LIN {X 0,Y 106.006,Z 264.737,A -85,B 0,C 180,E1 -28471.398,E2 -28471.398} C_VEL
LIN {X 0,Y 102.462,Z 273.009,A -85,B 0,C 180,E1 -28472.836,E2 -28472.836} C_VEL
LIN {X 0,Y 98.379,Z 281.013,A -85,B 0,C 180,E1 -28474.767,E2 -28474.767} C_VEL
LIN {X 0,Y 93.024,Z 289.74,A -85,B 0,C 180,E1 -28477.584,E2 -28477.584} C_VEL
LIN {X 0,Y 86.706,Z 298.118,A -85,B 0,C 180,E1 -28481.432,E2 -28481.432} C_VEL
LIN {X 0,Y 82.048,Z 303.608,A -85,B 0,C 180,E1 -28485.037,E2 -28485.037} C_VEL
LIN {X 0,Y 76.639,Z 309.153,A -85,B 0,C 180,E1 -28490.067,E2 -28490.067} C_VEL
LIN {X 0,Y 71.093,Z 314.313,A -85,B 0,C 180,E1 -28497.065,E2 -28497.065} C_VEL
LIN {X 0,Y 66.84,Z 318.102,A -85,B 0,C 180,E1 -28505.13,E2 -28505.13} C_VEL
LIN {X 0,Y 64.768,Z 319.84,A -85,B 0,C 180,E1 -28511.004,E2 -28511.004} C_VEL
LIN {X 0,Y 63.342,Z 321.084,A -85,B 0,C 180,E1 -28517.181,E2 -28517.181} C_VEL
LIN {X 0,Y 62.596,Z 321.855,A -85,B 0,C 180,E1 -28523.555,E2 -28523.555} C_VEL
LIN {X 0,Y 62.546,Z 322.148,A -85,B 0,C 180,E1 -28530.002,E2 -28530.002} C_VEL
LIN {X 0,Y 62.595,Z 321.84,A -85,B 0,C 180,E1 -28536.448,E2 -28536.448} C_VEL
LIN {X 0,Y 63.338,Z 321.04,A -85,B 0,C 180,E1 -28542.823,E2 -28542.823} C_VEL
LIN {X 0,Y 64.752,Z 319.768,A -85,B 0,C 180,E1 -28549.004,E2 -28549.004} C_VEL
LIN {X 0,Y 68.103,Z 316.843,A -85,B 0,C 180,E1 -28557.672,E2 -28557.672} C_VEL
LIN {X 0,Y 71.086,Z 314.178,A -85,B 0,C 180,E1 -28562.942,E2 -28562.942} C_VEL
LIN {X 0,Y 76.621,Z 308.98,A -85,B 0,C 180,E1 -28569.948,E2 -28569.948} C_VEL
LIN {X 0,Y 83.174,Z 302.123,A -85,B 0,C 180,E1 -28575.91,E2 -28575.91} C_VEL
LIN {X 0,Y 89.214,Z 294.637,A -85,B 0,C 180,E1 -28580.183,E2 -28580.183} C_VEL
LIN {X 0,Y 94.643,Z 286.803,A -85,B 0,C 180,E1 -28583.357,E2 -28583.357} C_VEL
LIN {X 0,Y 98.847,Z 279.71,A -85,B 0,C 180,E1 -28585.475,E2 -28585.475} C_VEL
LIN {X 0,Y 103.176,Z 270.972,A -85,B 0,C 180,E1 -28587.454,E2 -28587.454} C_VEL
LIN {X 0,Y 107.193,Z 260.903,A -85,B 0,C 180,E1 -28589.085,E2 -28589.085} C_VEL
LIN {X 0,Y 110.412,Z 249.756,A -85,B 0,C 180,E1 -28590.251,E2 -28590.251} C_VEL
LIN {X 0,Y 112.274,Z 240.076,A -85,B 0,C 180,E1 -28590.927,E2 -28590.927} C_VEL
LIN {X 0,Y 112.893,Z 234.742,A -85,B 0,C 180,E1 -28591.299,E2 -28591.299} C_VEL
LIN {X 0,Y 110.571,Z 229.113,A -85,B 0,C 180,E1 -28594.385,E2 -28594.385} C_VEL
LIN {X 0,Y 107.513,Z 222.914,A -85,B 0,C 180,E1 -28599.102,E2 -28599.102} C_VEL
LIN {X 0,Y 105.679,Z 219.605,A -85,B 0,C 180,E1 -28602.574,E2 -28602.574} C_VEL
LIN {X 0,Y 103.849,Z 216.166,A -85,B 0,C 180,E1 -28607.104,E2 -28607.104} C_VEL
LIN {X 0,Y 102.285,Z 213.382,A -85,B 0,C 180,E1 -28613.094,E2 -28613.094} C_VEL
LIN {X 0,Y 101.962,Z 211.83,A -85,B 0,C 180,E1 -28616.048,E2 -28616.048} C_VEL
LIN {X 0,Y 101.746,Z 211.461,A -85,B 0,C 180,E1 -28620,E2 -28620} C_VEL
LIN {X 0,Y 102.06,Z 212.11,A -85,B 0,C 180,E1 -28625.186,E2 -28625.186} C_VEL
LIN {X 0,Y 103.108,Z 215.279,A -85,B 0,C 180,E1 -28630.962,E2 -28630.962} C_VEL
LIN {X 0,Y 104.122,Z 216.678,A -85,B 0,C 180,E1 -28633.975,E2 -28633.975} C_VEL
LIN {X 0,Y 106.566,Z 221.249,A -85,B 0,C 180,E1 -28639.504,E2 -28639.504} C_VEL
LIN {X 0,Y 109.022,Z 225.911,A -85,B 0,C 180,E1 -28643.66,E2 -28643.66} C_VEL
LIN {X 0,Y 111.679,Z 231.652,A -85,B 0,C 180,E1 -28647.42,E2 -28647.42} C_VEL
LIN {X 0,Y 111.991,Z 233.692,A -85,B 0,C 180,E1 -28648.036,E2 -28648.036} C_VEL
LIN {X 0,Y 111.67,Z 236.769,A -85,B 0,C 180,E1 -28648.253,E2 -28648.253} C_VEL
LIN {X 0,Y 110.414,Z 241.191,A -85,B 0,C 180,E1 -28647.938,E2 -28647.938} C_VEL
LIN {X 0,Y 107.648,Z 248.027,A -85,B 0,C 180,E1 -28647.095,E2 -28647.095} C_VEL
LIN {X 0,Y 106.129,Z 252.208,A -85,B 0,C 180,E1 -28647.118,E2 -28647.118} C_VEL
LIN {X 0,Y 102.863,Z 261.996,A -85,B 0,C 180,E1 -28648.34,E2 -28648.34} C_VEL
LIN {X 0,Y 99.46,Z 270.01,A -85,B 0,C 180,E1 -28649.711,E2 -28649.711} C_VEL
LIN {X 0,Y 95.68,Z 277.368,A -85,B 0,C 180,E1 -28651.361,E2 -28651.361} C_VEL
LIN {X 0,Y 90.795,Z 285.27,A -85,B 0,C 180,E1 -28653.682,E2 -28653.682} C_VEL
LIN {X 0,Y 86.772,Z 290.94,A -85,B 0,C 180,E1 -28655.908,E2 -28655.908} C_VEL
LIN {X 0,Y 81.521,Z 297.279,A -85,B 0,C 180,E1 -28659.112,E2 -28659.112} C_VEL
LIN {X 0,Y 76.576,Z 302.546,A -85,B 0,C 180,E1 -28662.757,E2 -28662.757} C_VEL
LIN {X 0,Y 71.98,Z 306.943,A -85,B 0,C 180,E1 -28666.883,E2 -28666.883} C_VEL
LIN {X 0,Y 65.955,Z 312.112,A -85,B 0,C 180,E1 -28674.12,E2 -28674.12} C_VEL
LIN {X 0,Y 62.546,Z 314.761,A -85,B 0,C 180,E1 -28679.624,E2 -28679.624} C_VEL
LIN {X 0,Y 58.603,Z 317.66,A -85,B 0,C 180,E1 -28688.912,E2 -28688.912} C_VEL
LIN {X 0,Y 56.87,Z 318.92,A -85,B 0,C 180,E1 -28695.689,E2 -28695.689} C_VEL
LIN {X 0,Y 55.802,Z 319.711,A -85,B 0,C 180,E1 -28702.763,E2 -28702.763} C_VEL
LIN {X 0,Y 55.488,Z 320.012,A -85,B 0,C 180,E1 -28709.998,E2 -28709.998} C_VEL
LIN {X 0,Y 55.796,Z 319.73,A -85,B 0,C 180,E1 -28717.234,E2 -28717.234} C_VEL
LIN {X 0,Y 56.831,Z 318.976,A -85,B 0,C 180,E1 -28724.318,E2 -28724.318} C_VEL
LIN {X 0,Y 58.588,Z 317.754,A -85,B 0,C 180,E1 -28731.09,E2 -28731.09} C_VEL
LIN {X 0,Y 62.5,Z 314.894,A -85,B 0,C 180,E1 -28740.397,E2 -28740.397} C_VEL
LIN {X 0,Y 65.894,Z 312.287,A -85,B 0,C 180,E1 -28745.915,E2 -28745.915} C_VEL
LIN {X 0,Y 71.932,Z 307.164,A -85,B 0,C 180,E1 -28753.149,E2 -28753.149} C_VEL
LIN {X 0,Y 77.728,Z 301.649,A -85,B 0,C 180,E1 -28758.238,E2 -28758.238} C_VEL
LIN {X 0,Y 84.044,Z 294.711,A -85,B 0,C 180,E1 -28762.598,E2 -28762.598} C_VEL
LIN {X 0,Y 90.063,Z 286.746,A -85,B 0,C 180,E1 -28766.006,E2 -28766.006} C_VEL
LIN {X 0,Y 94.945,Z 279.15,A -85,B 0,C 180,E1 -28768.346,E2 -28768.346} C_VEL
LIN {X 0,Y 99.362,Z 270.874,A -85,B 0,C 180,E1 -28770.257,E2 -28770.257} C_VEL
LIN {X 0,Y 102.782,Z 263.051,A -85,B 0,C 180,E1 -28771.623,E2 -28771.623} C_VEL
LIN {X 0,Y 105.714,Z 254.557,A -85,B 0,C 180,E1 -28772.773,E2 -28772.773} C_VEL
LIN {X 0,Y 108.126,Z 245.305,A -85,B 0,C 180,E1 -28773.657,E2 -28773.657} C_VEL
LIN {X 0,Y 109.418,Z 238.026,A -85,B 0,C 180,E1 -28774.203,E2 -28774.203} C_VEL
LIN {X 0,Y 107.073,Z 231.956,A -85,B 0,C 180,E1 -28778.341,E2 -28778.341} C_VEL
LIN {X 0,Y 104.905,Z 227.419,A -85,B 0,C 180,E1 -28782.564,E2 -28782.564} C_VEL
LIN {X 0,Y 102.825,Z 223.047,A -85,B 0,C 180,E1 -28788.167,E2 -28788.167} C_VEL
LIN {X 0,Y 101.53,Z 220.472,A -85,B 0,C 180,E1 -28794.009,E2 -28794.009} C_VEL
LIN {X 0,Y 101.307,Z 218.967,A -85,B 0,C 180,E1 -28797.017,E2 -28797.017} C_VEL
LIN {X 0,Y 101.224,Z 218.755,A -85,B 0,C 180,E1 -28800.994,E2 -28800.994} C_VEL
LIN {X 0,Y 101.361,Z 219.335,A -85,B 0,C 180,E1 -28803.727,E2 -28803.727} C_VEL
LIN {X 0,Y 102.513,Z 222.681,A -85,B 0,C 180,E1 -28810.617,E2 -28810.617} C_VEL
LIN {X 0,Y 103.083,Z 223.715,A -85,B 0,C 180,E1 -28812.504,E2 -28812.504} C_VEL
LIN {X 0,Y 105.017,Z 227.64,A -85,B 0,C 180,E1 -28817.471,E2 -28817.471} C_VEL
LIN {X 0,Y 107.183,Z 232.16,A -85,B 0,C 180,E1 -28821.634,E2 -28821.634} C_VEL
LIN {X 0,Y 109.493,Z 238.014,A -85,B 0,C 180,E1 -28825.569,E2 -28825.569} C_VEL
LIN {X 0,Y 108.088,Z 246.375,A -85,B 0,C 180,E1 -28826.138,E2 -28826.138} C_VEL
LIN {X 0,Y 105.582,Z 255.84,A -85,B 0,C 180,E1 -28826.934,E2 -28826.934} C_VEL
LIN {X 0,Y 102.486,Z 264.614,A -85,B 0,C 180,E1 -28828.007,E2 -28828.007} C_VEL
LIN {X 0,Y 98.787,Z 272.886,A -85,B 0,C 180,E1 -28829.369,E2 -28829.369} C_VEL
LIN {X 0,Y 94.502,Z 280.888,A -85,B 0,C 180,E1 -28831.22,E2 -28831.22} C_VEL
LIN {X 0,Y 88.547,Z 290.089,A -85,B 0,C 180,E1 -28834.122,E2 -28834.122} C_VEL
LIN {X 0,Y 82.184,Z 297.992,A -85,B 0,C 180,E1 -28837.721,E2 -28837.721} C_VEL
LIN {X 0,Y 77.18,Z 303.481,A -85,B 0,C 180,E1 -28841.304,E2 -28841.304} C_VEL
LIN {X 0,Y 71.33,Z 309.026,A -85,B 0,C 180,E1 -28846.396,E2 -28846.396} C_VEL
LIN {X 0,Y 65.235,Z 314.185,A -85,B 0,C 180,E1 -28853.665,E2 -28853.665} C_VEL
LIN {X 0,Y 60.459,Z 317.975,A -85,B 0,C 180,E1 -28862.293,E2 -28862.293} C_VEL
LIN {X 0,Y 58.104,Z 319.712,A -85,B 0,C 180,E1 -28868.725,E2 -28868.725} C_VEL
LIN {X 0,Y 56.444,Z 320.956,A -85,B 0,C 180,E1 -28875.582,E2 -28875.582} C_VEL
LIN {X 0,Y 55.554,Z 321.727,A -85,B 0,C 180,E1 -28882.734,E2 -28882.734} C_VEL
LIN {X 0,Y 55.464,Z 322.02,A -85,B 0,C 180,E1 -28890.002,E2 -28890.002} C_VEL
LIN {X 0,Y 55.553,Z 321.712,A -85,B 0,C 180,E1 -28897.27,E2 -28897.27} C_VEL
LIN {X 0,Y 56.418,Z 320.911,A -85,B 0,C 180,E1 -28904.428,E2 -28904.428} C_VEL
LIN {X 0,Y 58.061,Z 319.638,A -85,B 0,C 180,E1 -28911.294,E2 -28911.294} C_VEL
LIN {X 0,Y 61.898,Z 316.713,A -85,B 0,C 180,E1 -28920.728,E2 -28920.728} C_VEL
LIN {X 0,Y 65.229,Z 314.048,A -85,B 0,C 180,E1 -28926.343,E2 -28926.343} C_VEL
LIN {X 0,Y 71.317,Z 308.85,A -85,B 0,C 180,E1 -28933.618,E2 -28933.618} C_VEL
LIN {X 0,Y 78.376,Z 301.991,A -85,B 0,C 180,E1 -28939.66,E2 -28939.66} C_VEL
LIN {X 0,Y 84.848,Z 294.506,A -85,B 0,C 180,E1 -28943.864,E2 -28943.864} C_VEL
LIN {X 0,Y 90.018,Z 287.496,A -85,B 0,C 180,E1 -28946.69,E2 -28946.69} C_VEL
LIN {X 0,Y 95.01,Z 279.578,A -85,B 0,C 180,E1 -28948.999,E2 -28948.999} C_VEL
LIN {X 0,Y 99.533,Z 270.838,A -85,B 0,C 180,E1 -28950.904,E2 -28950.904} C_VEL
LIN {X 0,Y 104.043,Z 259.898,A -85,B 0,C 180,E1 -28952.55,E2 -28952.55} C_VEL
LIN {X 0,Y 107.236,Z 248.925,A -85,B 0,C 180,E1 -28953.59,E2 -28953.59} C_VEL
LIN {X 0,Y 109.063,Z 239.444,A -85,B 0,C 180,E1 -28954.222,E2 -28954.222} C_VEL
LIN {X 0,Y 109.185,Z 237.645,A -85,B 0,C 180,E1 -28954.457,E2 -28954.457} C_VEL
LIN {X 0,Y 107.105,Z 232.42,A -85,B 0,C 180,E1 -28957.96,E2 -28957.96} C_VEL
LIN {X 0,Y 105.021,Z 227.961,A -85,B 0,C 180,E1 -28961.868,E2 -28961.868} C_VEL
LIN {X 0,Y 103.932,Z 225.805,A -85,B 0,C 180,E1 -28964.307,E2 -28964.307} C_VEL
LIN {X 0,Y 102.502,Z 222.849,A -85,B 0,C 180,E1 -28968.381,E2 -28968.381} C_VEL
LIN {X 0,Y 101.184,Z 219.881,A -85,B 0,C 180,E1 -28974.614,E2 -28974.614} C_VEL
LIN {X 0,Y 101.043,Z 218.843,A -85,B 0,C 180,E1 -28976.511,E2 -28976.511} C_VEL
LIN {X 0,Y 100.88,Z 218.518,A -85,B 0,C 180,E1 -28980,E2 -28980} C_VEL
LIN {X 0,Y 101.094,Z 219.124,A -85,B 0,C 180,E1 -28984.486,E2 -28984.486} C_VEL
LIN {X 0,Y 102.008,Z 222.171,A -85,B 0,C 180,E1 -28990.237,E2 -28990.237} C_VEL
LIN {X 0,Y 102.785,Z 223.36,A -85,B 0,C 180,E1 -28992.812,E2 -28992.812} C_VEL
LIN {X 0,Y 104.886,Z 227.692,A -85,B 0,C 180,E1 -28998.149,E2 -28998.149} C_VEL
LIN {X 0,Y 106.687,Z 231.486,A -85,B 0,C 180,E1 -29001.615,E2 -29001.615} C_VEL
LIN {X 0,Y 108.939,Z 237.118,A -85,B 0,C 180,E1 -29005.56,E2 -29005.56} C_VEL
LIN {X 0,Y 109.165,Z 237.748,A -85,B 0,C 180,E1 -29005.938,E2 -29005.938} C_VEL
LIN {X 0,Y 107.618,Z 246.129,A -85,B 0,C 180,E1 -29006.529,E2 -29006.529} C_VEL
LIN {X 0,Y 106.129,Z 252.208,A -85,B 0,C 180,E1 -29007.118,E2 -29007.118} C_VEL
LIN {X 0,Y 104.045,Z 257.981,A -85,B 0,C 180,E1 -29007.412,E2 -29007.412} C_VEL
LIN {X 0,Y 99.271,Z 266.842,A -85,B 0,C 180,E1 -29007.246,E2 -29007.246} C_VEL
LIN {X 0,Y 93.989,Z 274.963,A -85,B 0,C 180,E1 -29007.333,E2 -29007.333} C_VEL
LIN {X 0,Y 90.911,Z 279.638,A -85,B 0,C 180,E1 -29008.128,E2 -29008.128} C_VEL
LIN {X 0,Y 85.657,Z 287.439,A -85,B 0,C 180,E1 -29010.512,E2 -29010.512} C_VEL
LIN {X 0,Y 78.613,Z 295.995,A -85,B 0,C 180,E1 -29014.211,E2 -29014.211} C_VEL
LIN {X 0,Y 71.952,Z 302.677,A -85,B 0,C 180,E1 -29018.608,E2 -29018.608} C_VEL
LIN {X 0,Y 66.969,Z 307.073,A -85,B 0,C 180,E1 -29022.724,E2 -29022.724} C_VEL
LIN {X 0,Y 60.337,Z 312.242,A -85,B 0,C 180,E1 -29030.159,E2 -29030.159} C_VEL
LIN {X 0,Y 56.527,Z 314.89,A -85,B 0,C 180,E1 -29035.978,E2 -29035.978} C_VEL
LIN {X 0,Y 52.032,Z 317.789,A -85,B 0,C 180,E1 -29046.094,E2 -29046.094} C_VEL
LIN {X 0,Y 50.02,Z 319.049,A -85,B 0,C 180,E1 -29053.678,E2 -29053.678} C_VEL
LIN {X 0,Y 48.778,Z 319.84,A -85,B 0,C 180,E1 -29061.714,E2 -29061.714} C_VEL
LIN {X 0,Y 48.39,Z 320.141,A -85,B 0,C 180,E1 -29069.998,E2 -29069.998} C_VEL
LIN {X 0,Y 48.757,Z 319.859,A -85,B 0,C 180,E1 -29078.286,E2 -29078.286} C_VEL
LIN {X 0,Y 49.988,Z 319.104,A -85,B 0,C 180,E1 -29086.329,E2 -29086.329} C_VEL
LIN {X 0,Y 52.02,Z 317.882,A -85,B 0,C 180,E1 -29093.908,E2 -29093.908} C_VEL
LIN {X 0,Y 56.484,Z 315.021,A -85,B 0,C 180,E1 -29104.047,E2 -29104.047} C_VEL
LIN {X 0,Y 60.285,Z 312.414,A -85,B 0,C 180,E1 -29109.878,E2 -29109.878} C_VEL
LIN {X 0,Y 66.925,Z 307.291,A -85,B 0,C 180,E1 -29117.313,E2 -29117.313} C_VEL
LIN {X 0,Y 73.201,Z 301.776,A -85,B 0,C 180,E1 -29122.378,E2 -29122.378} C_VEL
LIN {X 0,Y 79.94,Z 294.837,A -85,B 0,C 180,E1 -29126.635,E2 -29126.635} C_VEL
LIN {X 0,Y 86.298,Z 286.871,A -85,B 0,C 180,E1 -29129.913,E2 -29129.913} C_VEL
LIN {X 0,Y 91.425,Z 279.274,A -85,B 0,C 180,E1 -29132.129,E2 -29132.129} C_VEL
LIN {X 0,Y 96.135,Z 270.791,A -85,B 0,C 180,E1 -29133.983,E2 -29133.983} C_VEL
LIN {X 0,Y 99.986,Z 262.221,A -85,B 0,C 180,E1 -29135.356,E2 -29135.356} C_VEL
LIN {X 0,Y 103.07,Z 253.413,A -85,B 0,C 180,E1 -29136.416,E2 -29136.416} C_VEL
LIN {X 0,Y 105.859,Z 242.498,A -85,B 0,C 180,E1 -29137.316,E2 -29137.316} C_VEL
LIN {X 0,Y 105.97,Z 241.214,A -85,B 0,C 180,E1 -29137.603,E2 -29137.603} C_VEL
LIN {X 0,Y 104.174,Z 236.115,A -85,B 0,C 180,E1 -29141.651,E2 -29141.651} C_VEL
LIN {X 0,Y 102.721,Z 232.517,A -85,B 0,C 180,E1 -29145.545,E2 -29145.545} C_VEL
LIN {X 0,Y 101.623,Z 229.837,A -85,B 0,C 180,E1 -29149.162,E2 -29149.162} C_VEL
LIN {X 0,Y 100.489,Z 227.015,A -85,B 0,C 180,E1 -29155.487,E2 -29155.487} C_VEL
LIN {X 0,Y 100.38,Z 225.926,A -85,B 0,C 180,E1 -29157.993,E2 -29157.993} C_VEL
LIN {X 0,Y 100.356,Z 225.825,A -85,B 0,C 180,E1 -29161.003,E2 -29161.003} C_VEL
LIN {X 0,Y 100.425,Z 226.32,A -85,B 0,C 180,E1 -29163.008,E2 -29163.008} C_VEL
LIN {X 0,Y 101.43,Z 229.596,A -85,B 0,C 180,E1 -29169.943,E2 -29169.943} C_VEL
LIN {X 0,Y 101.999,Z 231.005,A -85,B 0,C 180,E1 -29172.079,E2 -29172.079} C_VEL
LIN {X 0,Y 103.418,Z 234.077,A -85,B 0,C 180,E1 -29176.076,E2 -29176.076} C_VEL
LIN {X 0,Y 105.013,Z 238.252,A -85,B 0,C 180,E1 -29179.969,E2 -29179.969} C_VEL
LIN {X 0,Y 106.122,Z 241.412,A -85,B 0,C 180,E1 -29182.314,E2 -29182.314} C_VEL
LIN {X 0,Y 103.401,Z 253.172,A -85,B 0,C 180,E1 -29183.179,E2 -29183.179} C_VEL
LIN {X 0,Y 100.121,Z 262.617,A -85,B 0,C 180,E1 -29184.145,E2 -29184.145} C_VEL
LIN {X 0,Y 96.27,Z 271.26,A -85,B 0,C 180,E1 -29185.393,E2 -29185.393} C_VEL
LIN {X 0,Y 91.749,Z 279.531,A -85,B 0,C 180,E1 -29187.073,E2 -29187.073} C_VEL
LIN {X 0,Y 87.276,Z 286.418,A -85,B 0,C 180,E1 -29188.965,E2 -29188.965} C_VEL
LIN {X 0,Y 82.268,Z 292.98,A -85,B 0,C 180,E1 -29191.322,E2 -29191.322} C_VEL
LIN {X 0,Y 76.661,Z 299.287,A -85,B 0,C 180,E1 -29194.405,E2 -29194.405} C_VEL
LIN {X 0,Y 71.362,Z 304.528,A -85,B 0,C 180,E1 -29198.015,E2 -29198.015} C_VEL
LIN {X 0,Y 66.362,Z 308.899,A -85,B 0,C 180,E1 -29202.158,E2 -29202.158} C_VEL
LIN {X 0,Y 59.657,Z 314.058,A -85,B 0,C 180,E1 -29209.616,E2 -29209.616} C_VEL
LIN {X 0,Y 54.268,Z 317.847,A -85,B 0,C 180,E1 -29218.803,E2 -29218.803} C_VEL
LIN {X 0,Y 51.533,Z 319.584,A -85,B 0,C 180,E1 -29225.851,E2 -29225.851} C_VEL
LIN {X 0,Y 49.588,Z 320.827,A -85,B 0,C 180,E1 -29233.535,E2 -29233.535} C_VEL
LIN {X 0,Y 48.516,Z 321.598,A -85,B 0,C 180,E1 -29241.673,E2 -29241.673} C_VEL
LIN {X 0,Y 48.366,Z 321.891,A -85,B 0,C 180,E1 -29250.002,E2 -29250.002} C_VEL
LIN {X 0,Y 48.514,Z 321.583,A -85,B 0,C 180,E1 -29258.332,E2 -29258.332} C_VEL
LIN {X 0,Y 49.564,Z 320.782,A -85,B 0,C 180,E1 -29266.477,E2 -29266.477} C_VEL
LIN {X 0,Y 51.497,Z 319.509,A -85,B 0,C 180,E1 -29274.171,E2 -29274.171} C_VEL
LIN {X 0,Y 55.909,Z 316.584,A -85,B 0,C 180,E1 -29284.451,E2 -29284.451} C_VEL
LIN {X 0,Y 59.651,Z 313.918,A -85,B 0,C 180,E1 -29290.393,E2 -29290.393} C_VEL
LIN {X 0,Y 66.354,Z 308.72,A -85,B 0,C 180,E1 -29297.855,E2 -29297.855} C_VEL
LIN {X 0,Y 73.962,Z 301.86,A -85,B 0,C 180,E1 -29303.873,E2 -29303.873} C_VEL
LIN {X 0,Y 80.868,Z 294.375,A -85,B 0,C 180,E1 -29307.926,E2 -29307.926} C_VEL
LIN {X 0,Y 85.567,Z 288.439,A -85,B 0,C 180,E1 -29310.273,E2 -29310.273} C_VEL
LIN {X 0,Y 91.024,Z 280.307,A -85,B 0,C 180,E1 -29312.616,E2 -29312.616} C_VEL
LIN {X 0,Y 95.526,Z 272.207,A -85,B 0,C 180,E1 -29314.326,E2 -29314.326} C_VEL
LIN {X 0,Y 99.336,Z 263.798,A -85,B 0,C 180,E1 -29315.632,E2 -29315.632} C_VEL
LIN {X 0,Y 102.698,Z 254.431,A -85,B 0,C 180,E1 -29316.634,E2 -29316.634} C_VEL
LIN {X 0,Y 105.595,Z 243.006,A -85,B 0,C 180,E1 -29317.49,E2 -29317.49} C_VEL
LIN {X 0,Y 105.811,Z 241.005,A -85,B 0,C 180,E1 -29317.733,E2 -29317.733} C_VEL
LIN {X 0,Y 103.737,Z 235.205,A -85,B 0,C 180,E1 -29322.383,E2 -29322.383} C_VEL
LIN {X 0,Y 102.421,Z 232.296,A -85,B 0,C 180,E1 -29325.715,E2 -29325.715} C_VEL
LIN {X 0,Y 101.336,Z 229.664,A -85,B 0,C 180,E1 -29329.258,E2 -29329.258} C_VEL
LIN {X 0,Y 100.205,Z 226.801,A -85,B 0,C 180,E1 -29335.412,E2 -29335.412} C_VEL
LIN {X 0,Y 100.125,Z 225.904,A -85,B 0,C 180,E1 -29336.983,E2 -29336.983} C_VEL
LIN {X 0,Y 100.014,Z 225.573,A -85,B 0,C 180,E1 -29340,E2 -29340} C_VEL
LIN {X 0,Y 100.143,Z 226.145,A -85,B 0,C 180,E1 -29343.773,E2 -29343.773} C_VEL
LIN {X 0,Y 101.062,Z 229.288,A -85,B 0,C 180,E1 -29350.05,E2 -29350.05} C_VEL
LIN {X 0,Y 101.544,Z 230.264,A -85,B 0,C 180,E1 -29351.842,E2 -29351.842} C_VEL
LIN {X 0,Y 103.191,Z 233.997,A -85,B 0,C 180,E1 -29356.647,E2 -29356.647} C_VEL
LIN {X 0,Y 105.033,Z 238.917,A -85,B 0,C 180,E1 -29361.079,E2 -29361.079} C_VEL
LIN {X 0,Y 105.777,Z 241.123,A -85,B 0,C 180,E1 -29362.668,E2 -29362.668} C_VEL
LIN {X 0,Y 103.096,Z 252.341,A -85,B 0,C 180,E1 -29363.613,E2 -29363.613} C_VEL
LIN {X 0,Y 100.414,Z 260.361,A -85,B 0,C 180,E1 -29364.51,E2 -29364.51} C_VEL
LIN {X 0,Y 96.342,Z 269.736,A -85,B 0,C 180,E1 -29365.957,E2 -29365.957} C_VEL
LIN {X 0,Y 92.196,Z 277.5,A -85,B 0,C 180,E1 -29367.603,E2 -29367.603} C_VEL
LIN {X 0,Y 90.911,Z 279.638,A -85,B 0,C 180,E1 -29368.128,E2 -29368.128} C_VEL
LIN {X 0,Y 87.62,Z 284.322,A -85,B 0,C 180,E1 -29369.073,E2 -29369.073} C_VEL
LIN {X 0,Y 80.835,Z 291.459,A -85,B 0,C 180,E1 -29369.904,E2 -29369.904} C_VEL
LIN {X 0,Y 73.456,Z 297.901,A -85,B 0,C 180,E1 -29371.146,E2 -29371.146} C_VEL
LIN {X 0,Y 69.304,Z 301.497,A -85,B 0,C 180,E1 -29372.921,E2 -29372.921} C_VEL
LIN {X 0,Y 62.368,Z 307.203,A -85,B 0,C 180,E1 -29377.924,E2 -29377.924} C_VEL
LIN {X 0,Y 55.072,Z 312.372,A -85,B 0,C 180,E1 -29385.42,E2 -29385.42} C_VEL
LIN {X 0,Y 50.796,Z 315.02,A -85,B 0,C 180,E1 -29391.491,E2 -29391.491} C_VEL
LIN {X 0,Y 45.634,Z 317.919,A -85,B 0,C 180,E1 -29402.48,E2 -29402.48} C_VEL
LIN {X 0,Y 43.243,Z 319.178,A -85,B 0,C 180,E1 -29411.029,E2 -29411.029} C_VEL
LIN {X 0,Y 41.762,Z 319.969,A -85,B 0,C 180,E1 -29420.309,E2 -29420.309} C_VEL
LIN {X 0,Y 41.309,Z 320.269,A -85,B 0,C 180,E1 -29429.998,E2 -29429.998} C_VEL
LIN {X 0,Y 41.741,Z 319.987,A -85,B 0,C 180,E1 -29439.691,E2 -29439.691} C_VEL
LIN {X 0,Y 43.218,Z 319.232,A -85,B 0,C 180,E1 -29448.978,E2 -29448.978} C_VEL
LIN {X 0,Y 45.622,Z 318.009,A -85,B 0,C 180,E1 -29457.523,E2 -29457.523} C_VEL
LIN {X 0,Y 50.757,Z 315.149,A -85,B 0,C 180,E1 -29468.54,E2 -29468.54} C_VEL
LIN {X 0,Y 55.028,Z 312.541,A -85,B 0,C 180,E1 -29474.621,E2 -29474.621} C_VEL
LIN {X 0,Y 62.328,Z 307.418,A -85,B 0,C 180,E1 -29482.118,E2 -29482.118} C_VEL
LIN {X 0,Y 69.107,Z 301.902,A -85,B 0,C 180,E1 -29487.032,E2 -29487.032} C_VEL
LIN {X 0,Y 76.274,Z 294.962,A -85,B 0,C 180,E1 -29491.082,E2 -29491.082} C_VEL
LIN {X 0,Y 82.966,Z 286.996,A -85,B 0,C 180,E1 -29494.16,E2 -29494.16} C_VEL
LIN {X 0,Y 88.177,Z 279.653,A -85,B 0,C 180,E1 -29496.134,E2 -29496.134} C_VEL
LIN {X 0,Y 92.783,Z 271.805,A -85,B 0,C 180,E1 -29497.744,E2 -29497.744} C_VEL
LIN {X 0,Y 96.895,Z 263.187,A -85,B 0,C 180,E1 -29499.038,E2 -29499.038} C_VEL
LIN {X 0,Y 99.905,Z 255.172,A -85,B 0,C 180,E1 -29499.976,E2 -29499.976} C_VEL
LIN {X 0,Y 102.562,Z 245.801,A -85,B 0,C 180,E1 -29500.751,E2 -29500.751} C_VEL
LIN {X 0,Y 102.697,Z 244.87,A -85,B 0,C 180,E1 -29500.956,E2 -29500.956} C_VEL
LIN {X 0,Y 101.686,Z 240.83,A -85,B 0,C 180,E1 -29504.723,E2 -29504.723} C_VEL
LIN {X 0,Y 100.765,Z 238.323,A -85,B 0,C 180,E1 -29507.922,E2 -29507.922} C_VEL
LIN {X 0,Y 100.135,Z 236.377,A -85,B 0,C 180,E1 -29510.914,E2 -29510.914} C_VEL
LIN {X 0,Y 99.507,Z 233.043,A -85,B 0,C 180,E1 -29517.976,E2 -29517.976} C_VEL
LIN {X 0,Y 99.489,Z 232.892,A -85,B 0,C 180,E1 -29521.011,E2 -29521.011} C_VEL
LIN {X 0,Y 99.542,Z 234.081,A -85,B 0,C 180,E1 -29523.795,E2 -29523.795} C_VEL
LIN {X 0,Y 100.399,Z 237.011,A -85,B 0,C 180,E1 -29530.046,E2 -29530.046} C_VEL
LIN {X 0,Y 101.642,Z 240.555,A -85,B 0,C 180,E1 -29534.773,E2 -29534.773} C_VEL
LIN {X 0,Y 102.761,Z 244.481,A -85,B 0,C 180,E1 -29538.468,E2 -29538.468} C_VEL
LIN {X 0,Y 102.878,Z 245.149,A -85,B 0,C 180,E1 -29538.961,E2 -29538.961} C_VEL
LIN {X 0,Y 100.363,Z 254.384,A -85,B 0,C 180,E1 -29539.561,E2 -29539.561} C_VEL
LIN {X 0,Y 97.432,Z 262.495,A -85,B 0,C 180,E1 -29540.331,E2 -29540.331} C_VEL
LIN {X 0,Y 93.454,Z 271.137,A -85,B 0,C 180,E1 -29541.469,E2 -29541.469} C_VEL
LIN {X 0,Y 88.745,Z 279.403,A -85,B 0,C 180,E1 -29542.987,E2 -29542.987} C_VEL
LIN {X 0,Y 83.456,Z 287.115,A -85,B 0,C 180,E1 -29544.975,E2 -29544.975} C_VEL
LIN {X 0,Y 77.317,Z 294.561,A -85,B 0,C 180,E1 -29547.596,E2 -29547.596} C_VEL
LIN {X 0,Y 70.003,Z 301.991,A -85,B 0,C 180,E1 -29551.423,E2 -29551.423} C_VEL
LIN {X 0,Y 63.141,Z 307.814,A -85,B 0,C 180,E1 -29556.201,E2 -29556.201} C_VEL
LIN {X 0,Y 56.771,Z 312.407,A -85,B 0,C 180,E1 -29562.035,E2 -29562.035} C_VEL
LIN {X 0,Y 52.215,Z 315.396,A -85,B 0,C 180,E1 -29567.704,E2 -29567.704} C_VEL
LIN {X 0,Y 48.334,Z 317.719,A -85,B 0,C 180,E1 -29574.438,E2 -29574.438} C_VEL
LIN {X 0,Y 45.138,Z 319.456,A -85,B 0,C 180,E1 -29582.156,E2 -29582.156} C_VEL
LIN {X 0,Y 42.824,Z 320.699,A -85,B 0,C 180,E1 -29590.841,E2 -29590.841} C_VEL
LIN {X 0,Y 41.493,Z 321.47,A -85,B 0,C 180,E1 -29600.251,E2 -29600.251} C_VEL
LIN {X 0,Y 41.282,Z 321.763,A -85,B 0,C 180,E1 -29610.002,E2 -29610.002} C_VEL
LIN {X 0,Y 41.491,Z 321.455,A -85,B 0,C 180,E1 -29619.755,E2 -29619.755} C_VEL
LIN {X 0,Y 42.803,Z 320.653,A -85,B 0,C 180,E1 -29629.173,E2 -29629.173} C_VEL
LIN {X 0,Y 45.108,Z 319.379,A -85,B 0,C 180,E1 -29637.869,E2 -29637.869} C_VEL
LIN {X 0,Y 50.192,Z 316.454,A -85,B 0,C 180,E1 -29649.06,E2 -29649.06} C_VEL
LIN {X 0,Y 54.436,Z 313.788,A -85,B 0,C 180,E1 -29655.244,E2 -29655.244} C_VEL
LIN {X 0,Y 61.813,Z 308.59,A -85,B 0,C 180,E1 -29662.741,E2 -29662.741} C_VEL
LIN {X 0,Y 70.003,Z 301.729,A -85,B 0,C 180,E1 -29668.582,E2 -29668.582} C_VEL
LIN {X 0,Y 77.326,Z 294.243,A -85,B 0,C 180,E1 -29672.397,E2 -29672.397} C_VEL
LIN {X 0,Y 82.28,Z 288.308,A -85,B 0,C 180,E1 -29674.567,E2 -29674.567} C_VEL
LIN {X 0,Y 87.987,Z 280.175,A -85,B 0,C 180,E1 -29676.72,E2 -29676.72} C_VEL
LIN {X 0,Y 92.674,Z 272.074,A -85,B 0,C 180,E1 -29678.28,E2 -29678.28} C_VEL
LIN {X 0,Y 96.622,Z 263.663,A -85,B 0,C 180,E1 -29679.472,E2 -29679.472} C_VEL
LIN {X 0,Y 100.093,Z 254.295,A -85,B 0,C 180,E1 -29680.37,E2 -29680.37} C_VEL
LIN {X 0,Y 102.636,Z 244.758,A -85,B 0,C 180,E1 -29681.044,E2 -29681.044} C_VEL
LIN {X 0,Y 101.371,Z 240.338,A -85,B 0,C 180,E1 -29685.149,E2 -29685.149} C_VEL
LIN {X 0,Y 100.019,Z 236.421,A -85,B 0,C 180,E1 -29690.392,E2 -29690.392} C_VEL
LIN {X 0,Y 99.193,Z 232.839,A -85,B 0,C 180,E1 -29697.97,E2 -29697.97} C_VEL
LIN {X 0,Y 99.179,Z 232.806,A -85,B 0,C 180,E1 -29702.031,E2 -29702.031} C_VEL
LIN {X 0,Y 99.297,Z 234.407,A -85,B 0,C 180,E1 -29705.331,E2 -29705.331} C_VEL
LIN {X 0,Y 100.114,Z 236.827,A -85,B 0,C 180,E1 -29710.537,E2 -29710.537} C_VEL
LIN {X 0,Y 101.43,Z 240.637,A -85,B 0,C 180,E1 -29715.481,E2 -29715.481} C_VEL
LIN {X 0,Y 102.484,Z 244.693,A -85,B 0,C 180,E1 -29719.273,E2 -29719.273} C_VEL
LIN {X 0,Y 100.133,Z 253.468,A -85,B 0,C 180,E1 -29719.984,E2 -29719.984} C_VEL
LIN {X 0,Y 96.9,Z 262.368,A -85,B 0,C 180,E1 -29720.963,E2 -29720.963} C_VEL
LIN {X 0,Y 92.987,Z 270.777,A -85,B 0,C 180,E1 -29722.204,E2 -29722.204} C_VEL
LIN {X 0,Y 88.272,Z 279.002,A -85,B 0,C 180,E1 -29723.869,E2 -29723.869} C_VEL
LIN {X 0,Y 83.018,Z 286.552,A -85,B 0,C 180,E1 -29725.908,E2 -29725.908} C_VEL
LIN {X 0,Y 76.329,Z 294.599,A -85,B 0,C 180,E1 -29728.987,E2 -29728.987} C_VEL
LIN {X 0,Y 69.304,Z 301.497,A -85,B 0,C 180,E1 -29732.921,E2 -29732.921} C_VEL
LIN {X 0,Y 66.343,Z 303.771,A -85,B 0,C 180,E1 -29734.13,E2 -29734.13} C_VEL
LIN {X 0,Y 60.552,Z 307.131,A -85,B 0,C 180,E1 -29735.045,E2 -29735.045} C_VEL
LIN {X 0,Y 54.626,Z 310.127,A -85,B 0,C 180,E1 -29736.328,E2 -29736.328} C_VEL
LIN {X 0,Y 51.53,Z 311.749,A -85,B 0,C 180,E1 -29738.363,E2 -29738.363} C_VEL
LIN {X 0,Y 45.458,Z 315.149,A -85,B 0,C 180,E1 -29745.913,E2 -29745.913} C_VEL
LIN {X 0,Y 39.483,Z 318.047,A -85,B 0,C 180,E1 -29757.721,E2 -29757.721} C_VEL
LIN {X 0,Y 36.605,Z 319.306,A -85,B 0,C 180,E1 -29767.416,E2 -29767.416} C_VEL
LIN {X 0,Y 34.789,Z 320.097,A -85,B 0,C 180,E1 -29778.342,E2 -29778.342} C_VEL
LIN {X 0,Y 34.22,Z 320.397,A -85,B 0,C 180,E1 -29789.997,E2 -29789.997} C_VEL
LIN {X 0,Y 34.772,Z 320.115,A -85,B 0,C 180,E1 -29801.658,E2 -29801.658} C_VEL
LIN {X 0,Y 36.584,Z 319.36,A -85,B 0,C 180,E1 -29812.592,E2 -29812.592} C_VEL
LIN {X 0,Y 39.471,Z 318.137,A -85,B 0,C 180,E1 -29822.284,E2 -29822.284} C_VEL
LIN {X 0,Y 45.423,Z 315.276,A -85,B 0,C 180,E1 -29834.124,E2 -29834.124} C_VEL
LIN {X 0,Y 50.226,Z 312.668,A -85,B 0,C 180,E1 -29840.314,E2 -29840.314} C_VEL
LIN {X 0,Y 58.24,Z 307.545,A -85,B 0,C 180,E1 -29847.637,E2 -29847.637} C_VEL
LIN {X 0,Y 65.518,Z 302.028,A -85,B 0,C 180,E1 -29852.243,E2 -29852.243} C_VEL
LIN {X 0,Y 73.112,Z 295.088,A -85,B 0,C 180,E1 -29855.947,E2 -29855.947} C_VEL
LIN {X 0,Y 80.124,Z 287.122,A -85,B 0,C 180,E1 -29858.739,E2 -29858.739} C_VEL
LIN {X 0,Y 85.366,Z 280.073,A -85,B 0,C 180,E1 -29860.413,E2 -29860.413} C_VEL
LIN {X 0,Y 90.532,Z 271.559,A -85,B 0,C 180,E1 -29861.972,E2 -29861.972} C_VEL
LIN {X 0,Y 94.592,Z 263.31,A -85,B 0,C 180,E1 -29863.049,E2 -29863.049} C_VEL
LIN {X 0,Y 98.142,Z 253.998,A -85,B 0,C 180,E1 -29863.991,E2 -29863.991} C_VEL
LIN {X 0,Y 99.724,Z 248.67,A -85,B 0,C 180,E1 -29864.51,E2 -29864.51} C_VEL
LIN {X 0,Y 99.034,Z 245.307,A -85,B 0,C 180,E1 -29868.427,E2 -29868.427} C_VEL
LIN {X 0,Y 98.629,Z 243.127,A -85,B 0,C 180,E1 -29871.806,E2 -29871.806} C_VEL
LIN {X 0,Y 98.332,Z 239.919,A -85,B 0,C 180,E1 -29878.976,E2 -29878.976} C_VEL
LIN {X 0,Y 98.332,Z 239.998,A -85,B 0,C 180,E1 -29881.151,E2 -29881.151} C_VEL
LIN {X 0,Y 98.809,Z 243.779,A -85,B 0,C 180,E1 -29889.047,E2 -29889.047} C_VEL
LIN {X 0,Y 99.52,Z 247.016,A -85,B 0,C 180,E1 -29893.529,E2 -29893.529} C_VEL
LIN {X 0,Y 99.833,Z 248.649,A -85,B 0,C 180,E1 -29895.203,E2 -29895.203} C_VEL
LIN {X 0,Y 97.506,Z 256.345,A -85,B 0,C 180,E1 -29895.815,E2 -29895.815} C_VEL
LIN {X 0,Y 93.561,Z 266.121,A -85,B 0,C 180,E1 -29896.722,E2 -29896.722} C_VEL
LIN {X 0,Y 87.848,Z 276.818,A -85,B 0,C 180,E1 -29898.195,E2 -29898.195} C_VEL
LIN {X 0,Y 82.221,Z 285.066,A -85,B 0,C 180,E1 -29899.911,E2 -29899.911} C_VEL
LIN {X 0,Y 75.86,Z 292.728,A -85,B 0,C 180,E1 -29902.117,E2 -29902.117} C_VEL
LIN {X 0,Y 69.639,Z 299.035,A -85,B 0,C 180,E1 -29904.734,E2 -29904.734} C_VEL
LIN {X 0,Y 63.588,Z 304.274,A -85,B 0,C 180,E1 -29907.852,E2 -29907.852} C_VEL
LIN {X 0,Y 57.797,Z 308.645,A -85,B 0,C 180,E1 -29911.662,E2 -29911.662} C_VEL
LIN {X 0,Y 49.68,Z 313.803,A -85,B 0,C 180,E1 -29918.92,E2 -29918.92} C_VEL
LIN {X 0,Y 42.743,Z 317.591,A -85,B 0,C 180,E1 -29928.879,E2 -29928.879} C_VEL
LIN {X 0,Y 38.999,Z 319.328,A -85,B 0,C 180,E1 -29937.277,E2 -29937.277} C_VEL
LIN {X 0,Y 36.199,Z 320.571,A -85,B 0,C 180,E1 -29947.154,E2 -29947.154} C_VEL
LIN {X 0,Y 34.519,Z 321.341,A -85,B 0,C 180,E1 -29958.256,E2 -29958.256} C_VEL
LIN {X 0,Y 34.173,Z 321.635,A -85,B 0,C 180,E1 -29970.003,E2 -29970.003} C_VEL
LIN {X 0,Y 34.516,Z 321.326,A -85,B 0,C 180,E1 -29981.751,E2 -29981.751} C_VEL
LIN {X 0,Y 36.153,Z 320.524,A -85,B 0,C 180,E1 -29992.882,E2 -29992.882} C_VEL
LIN {X 0,Y 38.975,Z 319.25,A -85,B 0,C 180,E1 -30002.752,E2 -30002.752} C_VEL
LIN {X 0,Y 44.887,Z 316.324,A -85,B 0,C 180,E1 -30014.798,E2 -30014.798} C_VEL
LIN {X 0,Y 49.676,Z 313.658,A -85,B 0,C 180,E1 -30021.092,E2 -30021.092} C_VEL
LIN {X 0,Y 57.794,Z 308.46,A -85,B 0,C 180,E1 -30028.349,E2 -30028.349} C_VEL
LIN {X 0,Y 66.576,Z 301.598,A -85,B 0,C 180,E1 -30033.808,E2 -30033.808} C_VEL
LIN {X 0,Y 74.299,Z 294.112,A -85,B 0,C 180,E1 -30037.262,E2 -30037.262} C_VEL
LIN {X 0,Y 80.298,Z 287.115,A -85,B 0,C 180,E1 -30039.507,E2 -30039.507} C_VEL
LIN {X 0,Y 85.432,Z 280.043,A -85,B 0,C 180,E1 -30041.094,E2 -30041.094} C_VEL
LIN {X 0,Y 90.282,Z 271.94,A -85,B 0,C 180,E1 -30042.48,E2 -30042.48} C_VEL
LIN {X 0,Y 94.367,Z 263.529,A -85,B 0,C 180,E1 -30043.513,E2 -30043.513} C_VEL
LIN {X 0,Y 97.936,Z 254.159,A -85,B 0,C 180,E1 -30044.285,E2 -30044.285} C_VEL
LIN {X 0,Y 99.599,Z 248.433,A -85,B 0,C 180,E1 -30044.688,E2 -30044.688} C_VEL
LIN {X 0,Y 98.862,Z 245.06,A -85,B 0,C 180,E1 -30048.622,E2 -30048.622} C_VEL
LIN {X 0,Y 98.373,Z 242.742,A -85,B 0,C 180,E1 -30052.302,E2 -30052.302} C_VEL
LIN {X 0,Y 98.019,Z 239.734,A -85,B 0,C 180,E1 -30058.973,E2 -30058.973} C_VEL
LIN {X 0,Y 98.006,Z 239.983,A -85,B 0,C 180,E1 -30062.055,E2 -30062.055} C_VEL
LIN {X 0,Y 98.486,Z 243.616,A -85,B 0,C 180,E1 -30069.571,E2 -30069.571} C_VEL
LIN {X 0,Y 99.245,Z 247.118,A -85,B 0,C 180,E1 -30074.353,E2 -30074.353} C_VEL
LIN {X 0,Y 99.443,Z 248.648,A -85,B 0,C 180,E1 -30075.704,E2 -30075.704} C_VEL
LIN {X 0,Y 95.415,Z 260.629,A -85,B 0,C 180,E1 -30076.752,E2 -30076.752} C_VEL
LIN {X 0,Y 91.35,Z 269.412,A -85,B 0,C 180,E1 -30077.815,E2 -30077.815} C_VEL
LIN {X 0,Y 86.553,Z 277.757,A -85,B 0,C 180,E1 -30079.262,E2 -30079.262} C_VEL
LIN {X 0,Y 80.951,Z 285.665,A -85,B 0,C 180,E1 -30081.042,E2 -30081.042} C_VEL
LIN {X 0,Y 74.712,Z 293.031,A -85,B 0,C 180,E1 -30083.482,E2 -30083.482} C_VEL
LIN {X 0,Y 67.058,Z 300.497,A -85,B 0,C 180,E1 -30087.018,E2 -30087.018} C_VEL
LIN {X 0,Y 58.273,Z 307.333,A -85,B 0,C 180,E1 -30092.407,E2 -30092.407} C_VEL
LIN {X 0,Y 51.53,Z 311.749,A -85,B 0,C 180,E1 -30098.363,E2 -30098.363} C_VEL
LIN {X 0,Y 47.204,Z 314.074,A -85,B 0,C 180,E1 -30102.29,E2 -30102.29} C_VEL
LIN {X 0,Y 39.182,Z 317.051,A -85,B 0,C 180,E1 -30108.987,E2 -30108.987} C_VEL
LIN {X 0,Y 31.742,Z 319.123,A -85,B 0,C 180,E1 -30119.165,E2 -30119.165} C_VEL
LIN {X 0,Y 28.805,Z 319.845,A -85,B 0,C 180,E1 -30128.803,E2 -30128.803} C_VEL
LIN {X 0,Y 27.121,Z 320.526,A -85,B 0,C 180,E1 -30149.996,E2 -30149.996} C_VEL
LIN {X 0,Y 27.875,Z 320.243,A -85,B 0,C 180,E1 -30164.6,E2 -30164.6} C_VEL
LIN {X 0,Y 30.169,Z 319.488,A -85,B 0,C 180,E1 -30177.765,E2 -30177.765} C_VEL
LIN {X 0,Y 33.673,Z 318.265,A -85,B 0,C 180,E1 -30188.762,E2 -30188.762} C_VEL
LIN {X 0,Y 40.635,Z 315.404,A -85,B 0,C 180,E1 -30201.101,E2 -30201.101} C_VEL
LIN {X 0,Y 46.023,Z 312.795,A -85,B 0,C 180,E1 -30207.125,E2 -30207.125} C_VEL
LIN {X 0,Y 54.773,Z 307.672,A -85,B 0,C 180,E1 -30213.916,E2 -30213.916} C_VEL
LIN {X 0,Y 62.527,Z 302.155,A -85,B 0,C 180,E1 -30218.013,E2 -30218.013} C_VEL
LIN {X 0,Y 70.522,Z 295.213,A -85,B 0,C 180,E1 -30221.211,E2 -30221.211} C_VEL
LIN {X 0,Y 77.836,Z 287.246,A -85,B 0,C 180,E1 -30223.603,E2 -30223.603} C_VEL
LIN {X 0,Y 83.982,Z 279.129,A -85,B 0,C 180,E1 -30225.187,E2 -30225.187} C_VEL
LIN {X 0,Y 89.052,Z 270.857,A -85,B 0,C 180,E1 -30226.446,E2 -30226.446} C_VEL
LIN {X 0,Y 93.607,Z 261.559,A -85,B 0,C 180,E1 -30227.428,E2 -30227.428} C_VEL
LIN {X 0,Y 96.289,Z 254.516,A -85,B 0,C 180,E1 -30228.019,E2 -30228.019} C_VEL
LIN {X 0,Y 96.866,Z 252.529,A -85,B 0,C 180,E1 -30228.488,E2 -30228.488} C_VEL
LIN {X 0,Y 96.598,Z 249.609,A -85,B 0,C 180,E1 -30233.21,E2 -30233.21} C_VEL
LIN {X 0,Y 96.737,Z 246.708,A -85,B 0,C 180,E1 -30240,E2 -30240} C_VEL
LIN {X 0,Y 96.784,Z 250.391,A -85,B 0,C 180,E1 -30248.087,E2 -30248.087} C_VEL
LIN {X 0,Y 97.014,Z 252.314,A -85,B 0,C 180,E1 -30251.007,E2 -30251.007} C_VEL
LIN {X 0,Y 96.59,Z 254.029,A -85,B 0,C 180,E1 -30251.614,E2 -30251.614} C_VEL
LIN {X 0,Y 92.982,Z 263.302,A -85,B 0,C 180,E1 -30252.24,E2 -30252.24} C_VEL
LIN {X 0,Y 89.211,Z 270.943,A -85,B 0,C 180,E1 -30252.961,E2 -30252.961} C_VEL
LIN {X 0,Y 84.219,Z 279.154,A -85,B 0,C 180,E1 -30254.053,E2 -30254.053} C_VEL
LIN {X 0,Y 78.982,Z 286.298,A -85,B 0,C 180,E1 -30255.418,E2 -30255.418} C_VEL
LIN {X 0,Y 73.481,Z 292.602,A -85,B 0,C 180,E1 -30256.979,E2 -30256.979} C_VEL
LIN {X 0,Y 66.983,Z 298.909,A -85,B 0,C 180,E1 -30259.217,E2 -30259.217} C_VEL
LIN {X 0,Y 60.589,Z 304.147,A -85,B 0,C 180,E1 -30261.887,E2 -30261.887} C_VEL
LIN {X 0,Y 54.41,Z 308.518,A -85,B 0,C 180,E1 -30265.292,E2 -30265.292} C_VEL
LIN {X 0,Y 45.546,Z 313.675,A -85,B 0,C 180,E1 -30271.935,E2 -30271.935} C_VEL
LIN {X 0,Y 37.676,Z 317.464,A -85,B 0,C 180,E1 -30281.746,E2 -30281.746} C_VEL
LIN {X 0,Y 33.238,Z 319.2,A -85,B 0,C 180,E1 -30290.634,E2 -30290.634} C_VEL
LIN {X 0,Y 29.768,Z 320.443,A -85,B 0,C 180,E1 -30301.827,E2 -30301.827} C_VEL
LIN {X 0,Y 27.619,Z 321.213,A -85,B 0,C 180,E1 -30315.262,E2 -30315.262} C_VEL
LIN {X 0,Y 27.068,Z 321.506,A -85,B 0,C 180,E1 -30330.004,E2 -30330.004} C_VEL
LIN {X 0,Y 27.614,Z 321.198,A -85,B 0,C 180,E1 -30344.748,E2 -30344.748} C_VEL
LIN {X 0,Y 29.73,Z 320.395,A -85,B 0,C 180,E1 -30358.219,E2 -30358.219} C_VEL
LIN {X 0,Y 33.219,Z 319.121,A -85,B 0,C 180,E1 -30369.401,E2 -30369.401} C_VEL
LIN {X 0,Y 40.152,Z 316.195,A -85,B 0,C 180,E1 -30381.97,E2 -30381.97} C_VEL
LIN {X 0,Y 45.543,Z 313.528,A -85,B 0,C 180,E1 -30388.078,E2 -30388.078} C_VEL
LIN {X 0,Y 54.408,Z 308.33,A -85,B 0,C 180,E1 -30394.72,E2 -30394.72} C_VEL
LIN {X 0,Y 63.761,Z 301.468,A -85,B 0,C 180,E1 -30399.541,E2 -30399.541} C_VEL
LIN {X 0,Y 71.851,Z 293.981,A -85,B 0,C 180,E1 -30402.497,E2 -30402.497} C_VEL
LIN {X 0,Y 77.414,Z 287.832,A -85,B 0,C 180,E1 -30404.196,E2 -30404.196} C_VEL
LIN {X 0,Y 83.402,Z 279.911,A -85,B 0,C 180,E1 -30405.717,E2 -30405.717} C_VEL
LIN {X 0,Y 88.318,Z 271.968,A -85,B 0,C 180,E1 -30406.846,E2 -30406.846} C_VEL
LIN {X 0,Y 92.228,Z 264.227,A -85,B 0,C 180,E1 -30407.658,E2 -30407.658} C_VEL
LIN {X 0,Y 95.551,Z 256.068,A -85,B 0,C 180,E1 -30408.207,E2 -30408.207} C_VEL
LIN {X 0,Y 96.416,Z 253.573,A -85,B 0,C 180,E1 -30408.376,E2 -30408.376} C_VEL
LIN {X 0,Y 96.771,Z 252.085,A -85,B 0,C 180,E1 -30408.935,E2 -30408.935} C_VEL
LIN {X 0,Y 96.41,Z 249.398,A -85,B 0,C 180,E1 -30413.197,E2 -30413.197} C_VEL
LIN {X 0,Y 96.418,Z 246.609,A -85,B 0,C 180,E1 -30419.478,E2 -30419.478} C_VEL
LIN {X 0,Y 96.341,Z 246.953,A -85,B 0,C 180,E1 -30421.568,E2 -30421.568} C_VEL
LIN {X 0,Y 96.436,Z 250.103,A -85,B 0,C 180,E1 -30428.381,E2 -30428.381} C_VEL
LIN {X 0,Y 96.63,Z 252.175,A -85,B 0,C 180,E1 -30431.54,E2 -30431.54} C_VEL
LIN {X 0,Y 96.536,Z 252.817,A -85,B 0,C 180,E1 -30431.965,E2 -30431.965} C_VEL
LIN {X 0,Y 93.139,Z 261.818,A -85,B 0,C 180,E1 -30432.671,E2 -30432.671} C_VEL
LIN {X 0,Y 89.182,Z 269.999,A -85,B 0,C 180,E1 -30433.539,E2 -30433.539} C_VEL
LIN {X 0,Y 84.062,Z 278.508,A -85,B 0,C 180,E1 -30434.823,E2 -30434.823} C_VEL
LIN {X 0,Y 78.686,Z 285.796,A -85,B 0,C 180,E1 -30436.223,E2 -30436.223} C_VEL
LIN {X 0,Y 72.18,Z 293.163,A -85,B 0,C 180,E1 -30438.312,E2 -30438.312} C_VEL
LIN {X 0,Y 64.142,Z 300.628,A -85,B 0,C 180,E1 -30441.352,E2 -30441.352} C_VEL
LIN {X 0,Y 54.799,Z 307.463,A -85,B 0,C 180,E1 -30446.132,E2 -30446.132} C_VEL
LIN {X 0,Y 46.052,Z 312.631,A -85,B 0,C 180,E1 -30452.925,E2 -30452.925} C_VEL
LIN {X 0,Y 40.665,Z 315.278,A -85,B 0,C 180,E1 -30458.944,E2 -30458.944} C_VEL
LIN {X 0,Y 33.708,Z 318.176,A -85,B 0,C 180,E1 -30471.278,E2 -30471.278} C_VEL
LIN {X 0,Y 28.805,Z 319.845,A -85,B 0,C 180,E1 -30488.803,E2 -30488.803} C_VEL
LIN {X 0,Y 27.443,Z 320.255,A -85,B 0,C 180,E1 -30496.292,E2 -30496.292} C_VEL
LIN {X 0,Y 24.798,Z 320.55,A -85,B 0,C 180,E1 -30512.7,E2 -30512.7} C_VEL
LIN {X 0,Y 24.193,Z 319.816,A -85,B 0,C 180,E1 -30540.951,E2 -30540.951} C_VEL
LIN {X 0,Y 27.204,Z 318.828,A -85,B 0,C 180,E1 -30554.836,E2 -30554.836} C_VEL
LIN {X 0,Y 27.848,Z 318.553,A -85,B 0,C 180,E1 -30556.385,E2 -30556.385} C_VEL
LIN {X 0,Y 33.756,Z 316.677,A -85,B 0,C 180,E1 -30566.381,E2 -30566.381} C_VEL
LIN {X 0,Y 42.592,Z 312.922,A -85,B 0,C 180,E1 -30575.162,E2 -30575.162} C_VEL
LIN {X 0,Y 52.047,Z 307.798,A -85,B 0,C 180,E1 -30580.942,E2 -30580.942} C_VEL
LIN {X 0,Y 60.23,Z 302.282,A -85,B 0,C 180,E1 -30584.285,E2 -30584.285} C_VEL
LIN {X 0,Y 68.569,Z 295.339,A -85,B 0,C 180,E1 -30586.824,E2 -30586.824} C_VEL
LIN {X 0,Y 76.142,Z 287.371,A -85,B 0,C 180,E1 -30588.718,E2 -30588.718} C_VEL
LIN {X 0,Y 81.941,Z 279.997,A -85,B 0,C 180,E1 -30589.851,E2 -30589.851} C_VEL
LIN {X 0,Y 86.931,Z 272.262,A -85,B 0,C 180,E1 -30590.832,E2 -30590.832} C_VEL
LIN {X 0,Y 91.267,Z 263.988,A -85,B 0,C 180,E1 -30591.561,E2 -30591.561} C_VEL
LIN {X 0,Y 93.552,Z 258.905,A -85,B 0,C 180,E1 -30591.922,E2 -30591.922} C_VEL
LIN {X 0,Y 94.15,Z 257.045,A -85,B 0,C 180,E1 -30592.385,E2 -30592.385} C_VEL
LIN {X 0,Y 94.182,Z 255.486,A -85,B 0,C 180,E1 -30595.72,E2 -30595.72} C_VEL
LIN {X 0,Y 94.608,Z 253.709,A -85,B 0,C 180,E1 -30600,E2 -30600} C_VEL
LIN {X 0,Y 94.251,Z 256.899,A -85,B 0,C 180,E1 -30607.135,E2 -30607.135} C_VEL
LIN {X 0,Y 93.904,Z 258.137,A -85,B 0,C 180,E1 -30607.612,E2 -30607.612} C_VEL
LIN {X 0,Y 89.076,Z 268.761,A -85,B 0,C 180,E1 -30608.298,E2 -30608.298} C_VEL
LIN {X 0,Y 83.639,Z 277.799,A -85,B 0,C 180,E1 -30609.141,E2 -30609.141} C_VEL
LIN {X 0,Y 78.529,Z 284.816,A -85,B 0,C 180,E1 -30610.124,E2 -30610.124} C_VEL
LIN {X 0,Y 71.729,Z 292.477,A -85,B 0,C 180,E1 -30611.543,E2 -30611.543} C_VEL
LIN {X 0,Y 64.995,Z 298.783,A -85,B 0,C 180,E1 -30613.305,E2 -30613.305} C_VEL
LIN {X 0,Y 58.312,Z 304.021,A -85,B 0,C 180,E1 -30615.386,E2 -30615.386} C_VEL
LIN {X 0,Y 51.774,Z 308.391,A -85,B 0,C 180,E1 -30618.162,E2 -30618.162} C_VEL
LIN {X 0,Y 42.218,Z 313.548,A -85,B 0,C 180,E1 -30623.718,E2 -30623.718} C_VEL
LIN {X 0,Y 33.355,Z 317.336,A -85,B 0,C 180,E1 -30632.568,E2 -30632.568} C_VEL
LIN {X 0,Y 28.095,Z 319.072,A -85,B 0,C 180,E1 -30641.376,E2 -30641.376} C_VEL
LIN {X 0,Y 23.74,Z 320.315,A -85,B 0,C 180,E1 -30653.701,E2 -30653.701} C_VEL
LIN {X 0,Y 20.826,Z 321.085,A -85,B 0,C 180,E1 -30670.282,E2 -30670.282} C_VEL
LIN {X 0,Y 19.977,Z 321.378,A -85,B 0,C 180,E1 -30690.005,E2 -30690.005} C_VEL
LIN {X 0,Y 20.82,Z 321.069,A -85,B 0,C 180,E1 -30709.734,E2 -30709.734} C_VEL
LIN {X 0,Y 23.712,Z 320.266,A -85,B 0,C 180,E1 -30726.36,E2 -30726.36} C_VEL
LIN {X 0,Y 28.08,Z 318.992,A -85,B 0,C 180,E1 -30738.669,E2 -30738.669} C_VEL
LIN {X 0,Y 36.196,Z 316.065,A -85,B 0,C 180,E1 -30750.902,E2 -30750.902} C_VEL
LIN {X 0,Y 42.217,Z 313.398,A -85,B 0,C 180,E1 -30756.296,E2 -30756.296} C_VEL
LIN {X 0,Y 51.774,Z 308.2,A -85,B 0,C 180,E1 -30761.848,E2 -30761.848} C_VEL
LIN {X 0,Y 61.641,Z 301.337,A -85,B 0,C 180,E1 -30765.731,E2 -30765.731} C_VEL
LIN {X 0,Y 70.043,Z 293.849,A -85,B 0,C 180,E1 -30768.048,E2 -30768.048} C_VEL
LIN {X 0,Y 76.706,Z 286.59,A -85,B 0,C 180,E1 -30769.585,E2 -30769.585} C_VEL
LIN {X 0,Y 82.787,Z 278.546,A -85,B 0,C 180,E1 -30770.712,E2 -30770.712} C_VEL
LIN {X 0,Y 88.866,Z 268.521,A -85,B 0,C 180,E1 -30771.706,E2 -30771.706} C_VEL
LIN {X 0,Y 93.657,Z 257.904,A -85,B 0,C 180,E1 -30772.326,E2 -30772.326} C_VEL
LIN {X 0,Y 94.011,Z 256.618,A -85,B 0,C 180,E1 -30772.847,E2 -30772.847} C_VEL
LIN {X 0,Y 94.368,Z 253.397,A -85,B 0,C 180,E1 -30780,E2 -30780} C_VEL
LIN {X 0,Y 93.948,Z 255.986,A -85,B 0,C 180,E1 -30786.445,E2 -30786.445} C_VEL
LIN {X 0,Y 93.9,Z 256.738,A -85,B 0,C 180,E1 -30787.636,E2 -30787.636} C_VEL
LIN {X 0,Y 93.609,Z 257.788,A -85,B 0,C 180,E1 -30788.073,E2 -30788.073} C_VEL
LIN {X 0,Y 88.242,Z 269.347,A -85,B 0,C 180,E1 -30788.968,E2 -30788.968} C_VEL
LIN {X 0,Y 83.03,Z 277.918,A -85,B 0,C 180,E1 -30789.947,E2 -30789.947} C_VEL
LIN {X 0,Y 77.858,Z 284.908,A -85,B 0,C 180,E1 -30790.986,E2 -30790.986} C_VEL
LIN {X 0,Y 71.946,Z 291.596,A -85,B 0,C 180,E1 -30792.349,E2 -30792.349} C_VEL
LIN {X 0,Y 65.246,Z 297.931,A -85,B 0,C 180,E1 -30794.195,E2 -30794.195} C_VEL
LIN {X 0,Y 58.608,Z 303.197,A -85,B 0,C 180,E1 -30796.392,E2 -30796.392} C_VEL
LIN {X 0,Y 52.066,Z 307.593,A -85,B 0,C 180,E1 -30799.108,E2 -30799.108} C_VEL
LIN {X 0,Y 42.615,Z 312.761,A -85,B 0,C 180,E1 -30804.893,E2 -30804.893} C_VEL
LIN {X 0,Y 36.628,Z 315.407,A -85,B 0,C 180,E1 -30810.289,E2 -30810.289} C_VEL
LIN {X 0,Y 28.51,Z 318.305,A -85,B 0,C 180,E1 -30822.303,E2 -30822.303} C_VEL
LIN {X 0,Y 22.22,Z 320.003,A -85,B 0,C 180,E1 -30842.831,E2 -30842.831} C_VEL
LIN {X 0,Y 20.027,Z 320.654,A -85,B 0,C 180,E1 -30869.995,E2 -30869.995} C_VEL
LIN {X 0,Y 21.088,Z 320.371,A -85,B 0,C 180,E1 -30889.463,E2 -30889.463} C_VEL
LIN {X 0,Y 24.113,Z 319.616,A -85,B 0,C 180,E1 -30905.651,E2 -30905.651} C_VEL
LIN {X 0,Y 27.848,Z 318.553,A -85,B 0,C 180,E1 -30916.385,E2 -30916.385} C_VEL
LIN {X 0,Y 31.598,Z 317.357,A -85,B 0,C 180,E1 -30924.911,E2 -30924.911} C_VEL
LIN {X 0,Y 37.677,Z 314.639,A -85,B 0,C 180,E1 -30937.156,E2 -30937.156} C_VEL
LIN {X 0,Y 44.652,Z 311.052,A -85,B 0,C 180,E1 -30945.662,E2 -30945.662} C_VEL
LIN {X 0,Y 49.458,Z 308.332,A -85,B 0,C 180,E1 -30948.378,E2 -30948.378} C_VEL
LIN {X 0,Y 58.707,Z 302.408,A -85,B 0,C 180,E1 -30950.966,E2 -30950.966} C_VEL
LIN {X 0,Y 67.309,Z 295.465,A -85,B 0,C 180,E1 -30952.706,E2 -30952.706} C_VEL
LIN {X 0,Y 75.079,Z 287.496,A -85,B 0,C 180,E1 -30954.019,E2 -30954.019} C_VEL
LIN {X 0,Y 81.378,Z 279.576,A -85,B 0,C 180,E1 -30954.844,E2 -30954.844} C_VEL
LIN {X 0,Y 85.74,Z 272.985,A -85,B 0,C 180,E1 -30955.444,E2 -30955.444} C_VEL
LIN {X 0,Y 90.602,Z 263.889,A -85,B 0,C 180,E1 -30956.015,E2 -30956.015} C_VEL
LIN {X 0,Y 91.479,Z 261.942,A -85,B 0,C 180,E1 -30956.429,E2 -30956.429} C_VEL
LIN {X 0,Y 91.983,Z 260.587,A -85,B 0,C 180,E1 -30960,E2 -30960} C_VEL
LIN {X 0,Y 91.527,Z 262.005,A -85,B 0,C 180,E1 -30963.437,E2 -30963.437} C_VEL
LIN {X 0,Y 86.83,Z 271.218,A -85,B 0,C 180,E1 -30963.863,E2 -30963.863} C_VEL
LIN {X 0,Y 81.938,Z 278.905,A -85,B 0,C 180,E1 -30964.38,E2 -30964.38} C_VEL
LIN {X 0,Y 75.856,Z 286.736,A -85,B 0,C 180,E1 -30965.173,E2 -30965.173} C_VEL
LIN {X 0,Y 68.919,Z 294.057,A -85,B 0,C 180,E1 -30966.159,E2 -30966.159} C_VEL
LIN {X 0,Y 60.283,Z 301.486,A -85,B 0,C 180,E1 -30967.726,E2 -30967.726} C_VEL
LIN {X 0,Y 51.724,Z 307.306,A -85,B 0,C 180,E1 -30969.914,E2 -30969.914} C_VEL
LIN {X 0,Y 43.241,Z 311.898,A -85,B 0,C 180,E1 -30972.802,E2 -30972.802} C_VEL
LIN {X 0,Y 36.572,Z 314.884,A -85,B 0,C 180,E1 -30976.099,E2 -30976.099} C_VEL
LIN {X 0,Y 30.122,Z 317.207,A -85,B 0,C 180,E1 -30981.057,E2 -30981.057} C_VEL
LIN {X 0,Y 23.99,Z 318.944,A -85,B 0,C 180,E1 -30988.503,E2 -30988.503} C_VEL
LIN {X 0,Y 18.502,Z 320.186,A -85,B 0,C 180,E1 -31000.569,E2 -31000.569} C_VEL
LIN {X 0,Y 14.348,Z 320.957,A -85,B 0,C 180,E1 -31020.678,E2 -31020.678} C_VEL
LIN {X 0,Y 12.875,Z 321.249,A -85,B 0,C 180,E1 -31050.008,E2 -31050.008} C_VEL
LIN {X 0,Y 14.342,Z 320.94,A -85,B 0,C 180,E1 -31079.35,E2 -31079.35} C_VEL
LIN {X 0,Y 18.483,Z 320.137,A -85,B 0,C 180,E1 -31099.516,E2 -31099.516} C_VEL
LIN {X 0,Y 23.982,Z 318.862,A -85,B 0,C 180,E1 -31111.55,E2 -31111.55} C_VEL
LIN {X 0,Y 33.318,Z 315.935,A -85,B 0,C 180,E1 -31121.672,E2 -31121.672} C_VEL
LIN {X 0,Y 39.894,Z 313.268,A -85,B 0,C 180,E1 -31125.685,E2 -31125.685} C_VEL
LIN {X 0,Y 50.017,Z 308.07,A -85,B 0,C 180,E1 -31129.616,E2 -31129.616} C_VEL
LIN {X 0,Y 60.287,Z 301.207,A -85,B 0,C 180,E1 -31132.274,E2 -31132.274} C_VEL
LIN {X 0,Y 68.923,Z 293.718,A -85,B 0,C 180,E1 -31133.836,E2 -31133.836} C_VEL
LIN {X 0,Y 75.681,Z 286.534,A -85,B 0,C 180,E1 -31134.861,E2 -31134.861} C_VEL
LIN {X 0,Y 81.073,Z 279.645,A -85,B 0,C 180,E1 -31135.508,E2 -31135.508} C_VEL
LIN {X 0,Y 85.622,Z 272.704,A -85,B 0,C 180,E1 -31136.009,E2 -31136.009} C_VEL
LIN {X 0,Y 89.938,Z 264.664,A -85,B 0,C 180,E1 -31136.457,E2 -31136.457} C_VEL
LIN {X 0,Y 90.604,Z 263.231,A -85,B 0,C 180,E1 -31136.525,E2 -31136.525} C_VEL
LIN {X 0,Y 91.357,Z 261.48,A -85,B 0,C 180,E1 -31137.225,E2 -31137.225} C_VEL
LIN {X 0,Y 91.76,Z 260.307,A -85,B 0,C 180,E1 -31140,E2 -31140} C_VEL
LIN {X 0,Y 91.285,Z 261.546,A -85,B 0,C 180,E1 -31143.313,E2 -31143.313} C_VEL
LIN {X 0,Y 90.891,Z 262.503,A -85,B 0,C 180,E1 -31143.951,E2 -31143.951} C_VEL
LIN {X 0,Y 86.729,Z 270.667,A -85,B 0,C 180,E1 -31144.452,E2 -31144.452} C_VEL
LIN {X 0,Y 81.594,Z 278.772,A -85,B 0,C 180,E1 -31145.143,E2 -31145.143} C_VEL
LIN {X 0,Y 75.956,Z 286.059,A -85,B 0,C 180,E1 -31145.91,E2 -31145.91} C_VEL
LIN {X 0,Y 69.049,Z 293.424,A -85,B 0,C 180,E1 -31147.068,E2 -31147.068} C_VEL
LIN {X 0,Y 60.437,Z 300.889,A -85,B 0,C 180,E1 -31148.711,E2 -31148.711} C_VEL
LIN {X 0,Y 50.195,Z 307.722,A -85,B 0,C 180,E1 -31151.44,E2 -31151.44} C_VEL
LIN {X 0,Y 40.148,Z 312.89,A -85,B 0,C 180,E1 -31155.673,E2 -31155.673} C_VEL
LIN {X 0,Y 33.609,Z 315.537,A -85,B 0,C 180,E1 -31159.772,E2 -31159.772} C_VEL
LIN {X 0,Y 24.305,Z 318.435,A -85,B 0,C 180,E1 -31169.826,E2 -31169.826} C_VEL
LIN {X 0,Y 18.823,Z 319.693,A -85,B 0,C 180,E1 -31181.683,E2 -31181.683} C_VEL
LIN {X 0,Y 14.596,Z 320.482,A -85,B 0,C 180,E1 -31201.209,E2 -31201.209} C_VEL
LIN {X 0,Y 12.946,Z 320.782,A -85,B 0,C 180,E1 -31229.992,E2 -31229.992} C_VEL
LIN {X 0,Y 14.585,Z 320.5,A -85,B 0,C 180,E1 -31258.799,E2 -31258.799} C_VEL
LIN {X 0,Y 18.81,Z 319.744,A -85,B 0,C 180,E1 -31278.345,E2 -31278.345} C_VEL
LIN {X 0,Y 24.286,Z 318.521,A -85,B 0,C 180,E1 -31290.236,E2 -31290.236} C_VEL
LIN {X 0,Y 33.587,Z 315.659,A -85,B 0,C 180,E1 -31300.316,E2 -31300.316} C_VEL
LIN {X 0,Y 40.126,Z 313.05,A -85,B 0,C 180,E1 -31304.424,E2 -31304.424} C_VEL
LIN {X 0,Y 49.458,Z 308.332,A -85,B 0,C 180,E1 -31308.378,E2 -31308.378} C_VEL
LIN {X 0,Y 54.223,Z 305.452,A -85,B 0,C 180,E1 -31310.575,E2 -31310.575} C_VEL
LIN {X 0,Y 61.415,Z 300.2,A -85,B 0,C 180,E1 -31314.994,E2 -31314.994} C_VEL
LIN {X 0,Y 68.314,Z 294.207,A -85,B 0,C 180,E1 -31318.406,E2 -31318.406} C_VEL
LIN {X 0,Y 72.42,Z 290.099,A -85,B 0,C 180,E1 -31319.281,E2 -31319.281} C_VEL
LIN {X 0,Y 77.307,Z 284.565,A -85,B 0,C 180,E1 -31319.703,E2 -31319.703} C_VEL
LIN {X 0,Y 70.278,Z 292.225,A -85,B 0,C 180,E1 -31320.111,E2 -31320.111} C_VEL
LIN {X 0,Y 63.254,Z 298.53,A -85,B 0,C 180,E1 -31320.668,E2 -31320.668} C_VEL
LIN {X 0,Y 56.236,Z 303.767,A -85,B 0,C 180,E1 -31321.284,E2 -31321.284} C_VEL
LIN {X 0,Y 49.231,Z 308.136,A -85,B 0,C 180,E1 -31322.223,E2 -31322.223} C_VEL
LIN {X 0,Y 38.751,Z 313.293,A -85,B 0,C 180,E1 -31324.098,E2 -31324.098} C_VEL
LIN {X 0,Y 28.352,Z 317.079,A -85,B 0,C 180,E1 -31327.482,E2 -31327.482} C_VEL
LIN {X 0,Y 21.523,Z 318.816,A -85,B 0,C 180,E1 -31331.612,E2 -31331.612} C_VEL
LIN {X 0,Y 14.887,Z 320.058,A -85,B 0,C 180,E1 -31339.253,E2 -31339.253} C_VEL
LIN {X 0,Y 8.861,Z 320.828,A -85,B 0,C 180,E1 -31357.54,E2 -31357.54} C_VEL
LIN {X 0,Y 5.767,Z 321.121,A -85,B 0,C 180,E1 -31410.017,E2 -31410.017} C_VEL
LIN {X 0,Y 8.858,Z 320.812,A -85,B 0,C 180,E1 -31462.52,E2 -31462.52} C_VEL
LIN {X 0,Y 14.88,Z 320.008,A -85,B 0,C 180,E1 -31480.858,E2 -31480.858} C_VEL
LIN {X 0,Y 21.522,Z 318.733,A -85,B 0,C 180,E1 -31488.444,E2 -31488.444} C_VEL
LIN {X 0,Y 31.806,Z 315.805,A -85,B 0,C 180,E1 -31493.936,E2 -31493.936} C_VEL
LIN {X 0,Y 38.754,Z 313.139,A -85,B 0,C 180,E1 -31495.916,E2 -31495.916} C_VEL
LIN {X 0,Y 49.234,Z 307.939,A -85,B 0,C 180,E1 -31497.786,E2 -31497.786} C_VEL
LIN {X 0,Y 59.748,Z 301.076,A -85,B 0,C 180,E1 -31499.024,E2 -31499.024} C_VEL
LIN {X 0,Y 67.659,Z 294.427,A -85,B 0,C 180,E1 -31499.696,E2 -31499.696} C_VEL
LIN {X 0,Y 73.796,Z 288.243,A -85,B 0,C 180,E1 -31500.124,E2 -31500.124} C_VEL
LIN {X 0,Y 77.312,Z 284.151,A -85,B 0,C 180,E1 -31500.439,E2 -31500.439} C_VEL
LIN {X 0,Y 70.292,Z 291.858,A -85,B 0,C 180,E1 -31500.981,E2 -31500.981} C_VEL
LIN {X 0,Y 63.279,Z 298.193,A -85,B 0,C 180,E1 -31501.632,E2 -31501.632} C_VEL
LIN {X 0,Y 56.275,Z 303.458,A -85,B 0,C 180,E1 -31502.392,E2 -31502.392} C_VEL
LIN {X 0,Y 49.281,Z 307.852,A -85,B 0,C 180,E1 -31503.331,E2 -31503.331} C_VEL
LIN {X 0,Y 38.835,Z 313.02,A -85,B 0,C 180,E1 -31505.509,E2 -31505.509} C_VEL
LIN {X 0,Y 31.915,Z 315.666,A -85,B 0,C 180,E1 -31507.695,E2 -31507.695} C_VEL
LIN {X 0,Y 21.67,Z 318.564,A -85,B 0,C 180,E1 -31513.333,E2 -31513.333} C_VEL
LIN {X 0,Y 15.062,Z 319.822,A -85,B 0,C 180,E1 -31521.046,E2 -31521.046} C_VEL
LIN {X 0,Y 9.051,Z 320.611,A -85,B 0,C 180,E1 -31539.041,E2 -31539.041} C_VEL
LIN {X 0,Y 5.874,Z 320.91,A -85,B 0,C 180,E1 -31589.983,E2 -31589.983} C_VEL
LIN {X 0,Y 9.042,Z 320.628,A -85,B 0,C 180,E1 -31640.989,E2 -31640.989} C_VEL
LIN {X 0,Y 15.054,Z 319.872,A -85,B 0,C 180,E1 -31659,E2 -31659} C_VEL
LIN {X 0,Y 21.66,Z 318.648,A -85,B 0,C 180,E1 -31666.741,E2 -31666.741} C_VEL
LIN {X 0,Y 31.902,Z 315.786,A -85,B 0,C 180,E1 -31672.432,E2 -31672.432} C_VEL
LIN {X 0,Y 38.826,Z 313.177,A -85,B 0,C 180,E1 -31674.584,E2 -31674.584} C_VEL
LIN {X 0,Y 49.274,Z 308.052,A -85,B 0,C 180,E1 -31676.734,E2 -31676.734} C_VEL
LIN {X 0,Y 58.018,Z 302.535,A -85,B 0,C 180,E1 -31677.904,E2 -31677.904} C_VEL
LIN {X 0,Y 67.908,Z 294.51,A -85,B 0,C 180,E1 -31678.894,E2 -31678.894} C_VEL
LIN {X 0,Y 72.42,Z 290.099,A -85,B 0,C 180,E1 -31679.281,E2 -31679.281} C_VEL
LIN {X 0,Y 75.859,Z 291.474,A -85,B 0,C 180,E1 -31679.512,E2 -31679.512} C_VEL
LIN {X 0,Y 75.859,Z 600,A -85,B 0,C 180,E1 -31679.512,E2 -31679.512} C_VEL
LIN {X 0,Y 75.859,Z 600,A -85,B 0,C 180,E1 -31679.512,E2 -31679.512}

QRS_NEXT_CUT()

QRS_NEXT()
QRS_HOME()

END
